FUNCTION_BLOCK FBME_E_SR
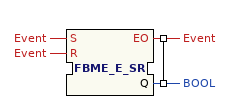
  EVENT_INPUT
    S;
    R;
  END_EVENT
  EVENT_OUTPUT
    EO WITH Q;
  END_EVENT
  VAR_OUTPUT
    Q : BOOL;
  END_VAR
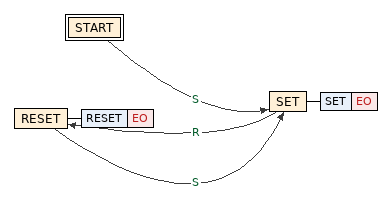
  EC_STATES
    START;
    SET : SET -> EO;
    RESET : RESET -> EO;
  END_STATES
  EC_TRANSITIONS
    START TO SET := S;
    SET TO RESET := R;
    RESET TO SET := S;
  END_TRANSITIONS
  ALGORITHM SET IN ST:
Q := TRUE;
  END_ALGORITHM
  ALGORITHM RESET IN ST:
Q := FALSE;
  END_ALGORITHM
END_FUNCTION_BLOCK
